RoboDK station: GA KUKA.rdk

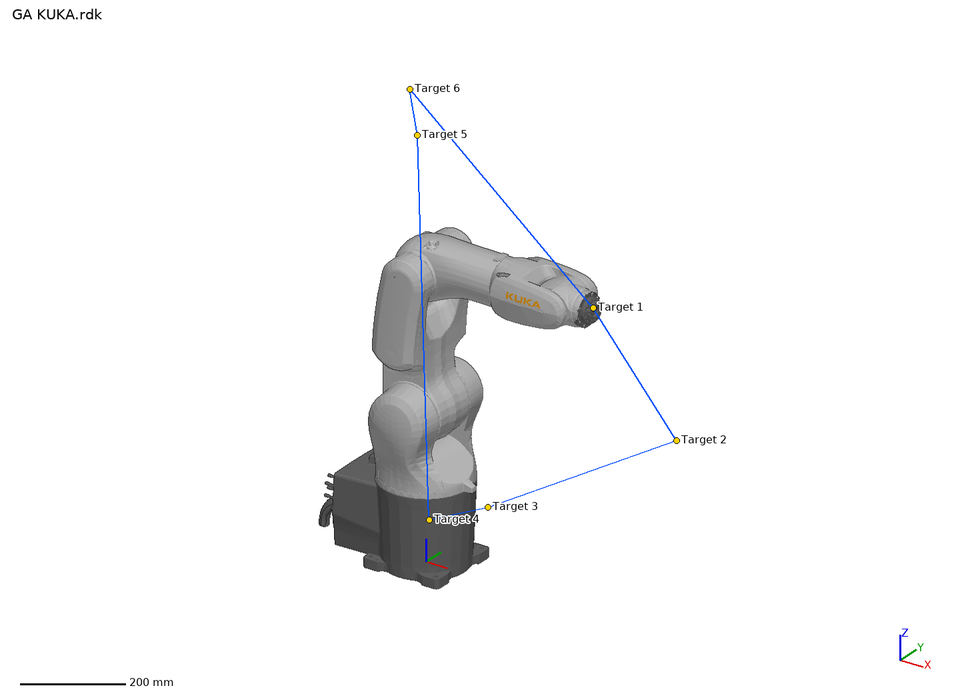
[picture v0: the station drawn from its stored meshes, robots at their saved joint values, targets as dots, program paths as lines]
Station New Station (1) (saved by RoboDK 5.5.4). Poses are relative to the parent item; angles as X-Y-Z fixed-axis rotations.
  - frame KUKA KR 4 R600 Base at (0, 0, 0) mm
    - robot KUKA KR 4 R600: 6 axes, payload 4.63 kg, reach 601 mm, repeatability 0.015 mm, weight 24 kg
        modified DH rows (alpha deg, a mm, theta deg, d mm): 0, 0, 0, 330; -90, 0, 0, 0; 0, 290, -90, 0; -90, 20, 0, 310; 90, 0, 0, 0; -90, 0, 180, 75
        joint limits [-170, -195, -115, -185, -120, -350] to [170, 40, 150, 180, 120, 350]; home [0, -90, 90, 0, 0, 0]; saved at [0, -88.99, 90, 0, 0, 0]
    - target Target 1 (Cartesian target) at (385, 0, 640) mm, rotated rx 0 ry 90 rz 0 deg; joints [0, -90, 90, 0, 0, 0] of KUKA KR 4 R600
    - target Target 2 (joint target) at (577.1, 0, 415.66) mm, rotated rx -179.95 ry 1.27 rz 2.38 deg; joints [0, -15.47, 3.61, 0, 103.132, -177.617] of KUKA KR 4 R600
    - target Target 3 (joint target) at (201.51, -83.66, 203.67) mm, rotated rx -93.47 ry 63.83 rz -117.14 deg; joints [21.772, -36.669, 147.078, 177.617, 108.862, -154.698] of KUKA KR 4 R600
    - target Target 4 (joint target) at (147.7, -200.48, 209.13) mm, rotated rx 75.11 ry 14.37 rz 153.57 deg; joints [65.89, -34.95, 118.373, 131.78, -108.862, -80.214] of KUKA KR 4 R600
    - target Target 5 (joint target) at (9.16, -41.91, 914.03) mm, rotated rx -101.97 ry -72.86 rz 30.16 deg; joints [-106.387, -99.121, -0.516, 177.617, -103.132, -17.189] of KUKA KR 4 R600
    - target Target 6 (joint target) at (-70.05, 46.68, 953.95) mm, rotated rx 68.49 ry 2.38 rz -156.4 deg; joints [-22.248, -99.694, 14.209, 85.943, -68.755, 97.403] of KUKA KR 4 R600
  - program Prog1 (8 instructions, listed below)
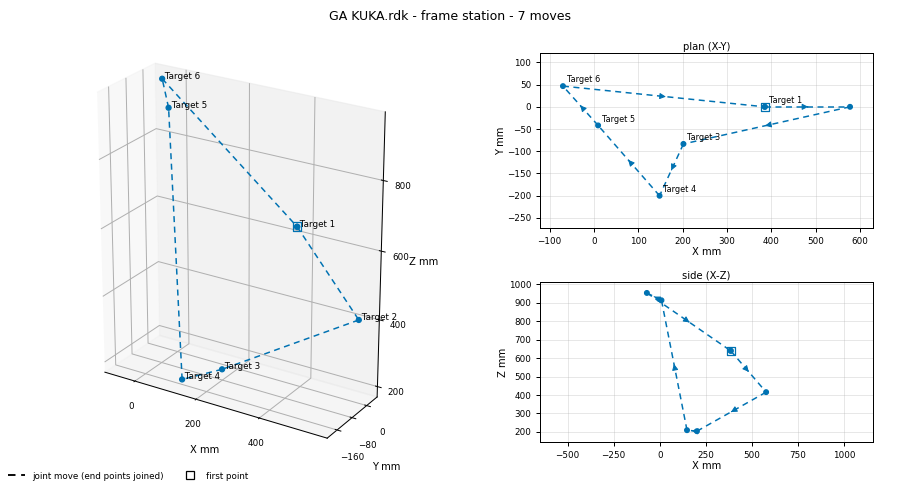
[picture p0: tool path of GA KUKA.rdk in frame station, 7 of 7 moves have a stored position in this frame; points joined in program order, loops and branches not executed]

--- program Prog1 (robot KUKA KR 4 R600) ---
  Set Ref.: KUKA KR 4 R600 Base
  MoveJ (Target 1)
  MoveJ (Target 2)
  MoveJ (Target 3)
  MoveJ (Target 4)
  MoveJ (Target 5)
  MoveJ (Target 6)
  MoveJ (Target 1)
